REGION Network 11: Output Feedback
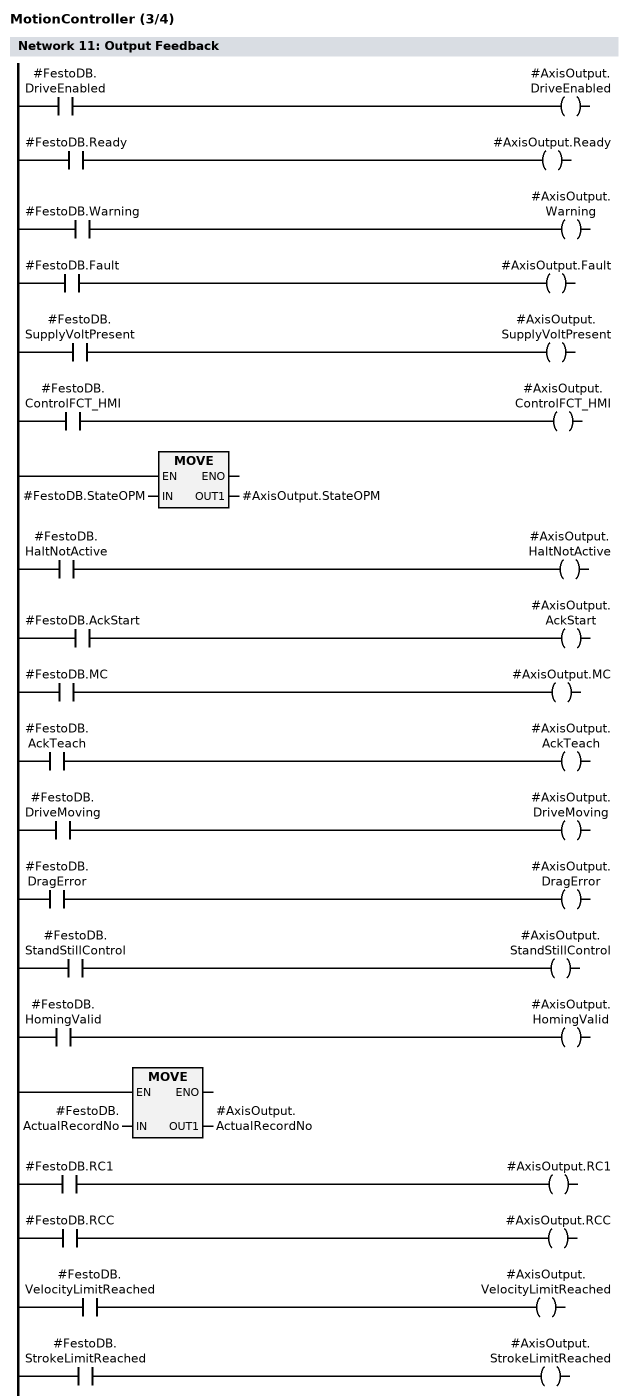
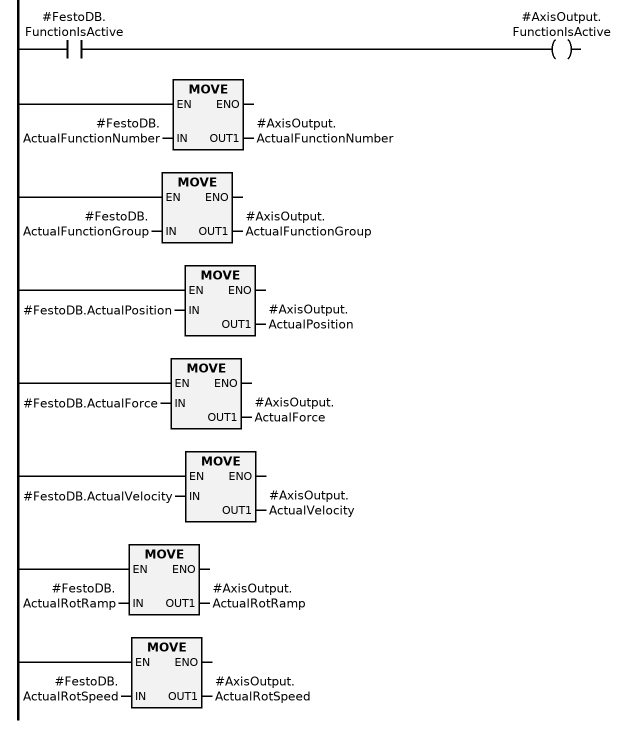
   RUNG wire#powerrail
      Contact( #FestoDB.DriveEnabled )
      Coil( #AxisOutput.DriveEnabled )
   END_RUNG
   RUNG wire#powerrail
      Contact( #FestoDB.Ready )
      Coil( #AxisOutput.Ready )
   END_RUNG
   RUNG wire#powerrail
      Contact( #FestoDB.Warning )
      Coil( #AxisOutput.Warning )
   END_RUNG
   RUNG wire#powerrail
      Contact( #FestoDB.Fault )
      Coil( #AxisOutput.Fault )
   END_RUNG
   RUNG wire#powerrail
      Contact( #FestoDB.SupplyVoltPresent )
      Coil( #AxisOutput.SupplyVoltPresent )
   END_RUNG
   RUNG wire#powerrail
      Contact( #FestoDB.ControlFCT_HMI )
      Coil( #AxisOutput.ControlFCT_HMI )
   END_RUNG
   RUNG wire#powerrail
      Move(in := #FestoDB.StateOPM, out1 => #AxisOutput.StateOPM)
   END_RUNG
   RUNG wire#powerrail
      Contact( #FestoDB.HaltNotActive )
      Coil( #AxisOutput.HaltNotActive )
   END_RUNG
   RUNG wire#powerrail
      Contact( #FestoDB.AckStart )
      Coil( #AxisOutput.AckStart )
   END_RUNG
   RUNG wire#powerrail
      Contact( #FestoDB.MC )
      Coil( #AxisOutput.MC )
   END_RUNG
   RUNG wire#powerrail
      Contact( #FestoDB.AckTeach )
      Coil( #AxisOutput.AckTeach )
   END_RUNG
   RUNG wire#powerrail
      Contact( #FestoDB.DriveMoving )
      Coil( #AxisOutput.DriveMoving )
   END_RUNG
   RUNG wire#powerrail
      Contact( #FestoDB.DragError )
      Coil( #AxisOutput.DragError )
   END_RUNG
   RUNG wire#powerrail
      Contact( #FestoDB.StandStillControl )
      Coil( #AxisOutput.StandStillControl )
   END_RUNG
   RUNG wire#powerrail
      Contact( #FestoDB.HomingValid )
      Coil( #AxisOutput.HomingValid )
   END_RUNG
   RUNG wire#powerrail
      Move(in := #FestoDB.ActualRecordNo, out1 => #AxisOutput.ActualRecordNo)
   END_RUNG
   RUNG wire#powerrail
      Contact( #FestoDB.RC1 )
      Coil( #AxisOutput.RC1 )
   END_RUNG
   RUNG wire#powerrail
      Contact( #FestoDB.RCC )
      Coil( #AxisOutput.RCC )
   END_RUNG
   RUNG wire#powerrail
      Contact( #FestoDB.VelocityLimitReached )
      Coil( #AxisOutput.VelocityLimitReached )
   END_RUNG
   RUNG wire#powerrail
      Contact( #FestoDB.StrokeLimitReached )
      Coil( #AxisOutput.StrokeLimitReached )
   END_RUNG
   RUNG wire#powerrail
      Contact( #FestoDB.FunctionIsActive )
      Coil( #AxisOutput.FunctionIsActive )
   END_RUNG
   RUNG wire#powerrail
      Move(in := #FestoDB.ActualFunctionNumber, out1 => #AxisOutput.ActualFunctionNumber)
   END_RUNG
   RUNG wire#powerrail
      Move(in := #FestoDB.ActualFunctionGroup, out1 => #AxisOutput.ActualFunctionGroup)
   END_RUNG
   RUNG wire#powerrail
      Move(in := #FestoDB.ActualPosition, out1 => #AxisOutput.ActualPosition)
   END_RUNG
   RUNG wire#powerrail
      Move(in := #FestoDB.ActualForce, out1 => #AxisOutput.ActualForce)
   END_RUNG
   RUNG wire#powerrail
      Move(in := #FestoDB.ActualVelocity, out1 => #AxisOutput.ActualVelocity)
   END_RUNG
   RUNG wire#powerrail
      Move(in := #FestoDB.ActualRotRamp, out1 => #AxisOutput.ActualRotRamp)
   END_RUNG
   RUNG wire#powerrail
      Move(in := #FestoDB.ActualRotSpeed, out1 => #AxisOutput.ActualRotSpeed)
   END_RUNG
   // the same network as SCL:
   #AxisOutput.DriveEnabled := #FestoDB.DriveEnabled;
   #AxisOutput.Ready := #FestoDB.Ready;
   #AxisOutput.Warning := #FestoDB.Warning;
   #AxisOutput.Fault := #FestoDB.Fault;
   #AxisOutput.SupplyVoltPresent := #FestoDB.SupplyVoltPresent;
   #AxisOutput.ControlFCT_HMI := #FestoDB.ControlFCT_HMI;
   #AxisOutput.StateOPM := #FestoDB.StateOPM;
   #AxisOutput.HaltNotActive := #FestoDB.HaltNotActive;
   #AxisOutput.AckStart := #FestoDB.AckStart;
   #AxisOutput.MC := #FestoDB.MC;
   #AxisOutput.AckTeach := #FestoDB.AckTeach;
   #AxisOutput.DriveMoving := #FestoDB.DriveMoving;
   #AxisOutput.DragError := #FestoDB.DragError;
   #AxisOutput.StandStillControl := #FestoDB.StandStillControl;
   #AxisOutput.HomingValid := #FestoDB.HomingValid;
   #AxisOutput.ActualRecordNo := #FestoDB.ActualRecordNo;
   #AxisOutput.RC1 := #FestoDB.RC1;
   #AxisOutput.RCC := #FestoDB.RCC;
   #AxisOutput.VelocityLimitReached := #FestoDB.VelocityLimitReached;
   #AxisOutput.StrokeLimitReached := #FestoDB.StrokeLimitReached;
   #AxisOutput.FunctionIsActive := #FestoDB.FunctionIsActive;
   #AxisOutput.ActualFunctionNumber := #FestoDB.ActualFunctionNumber;
   #AxisOutput.ActualFunctionGroup := #FestoDB.ActualFunctionGroup;
   #AxisOutput.ActualPosition := #FestoDB.ActualPosition;
   #AxisOutput.ActualForce := #FestoDB.ActualForce;
   #AxisOutput.ActualVelocity := #FestoDB.ActualVelocity;
   #AxisOutput.ActualRotRamp := #FestoDB.ActualRotRamp;
   #AxisOutput.ActualRotSpeed := #FestoDB.ActualRotSpeed;
END_REGION

REGION Network 12: TargetReached
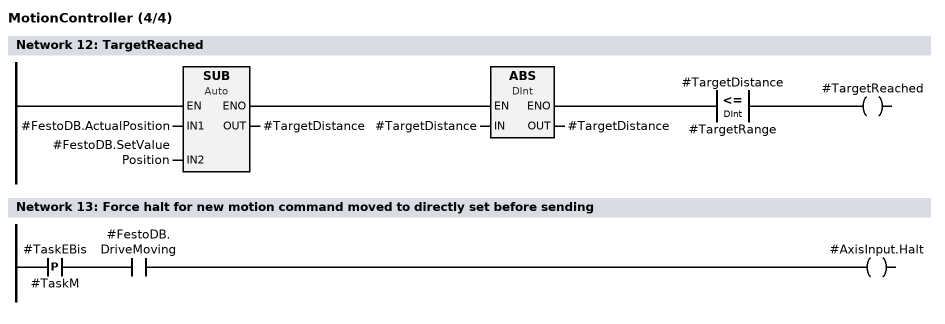
   RUNG wire#powerrail
      Sub(in1 := #FestoDB.ActualPosition, in2 := #FestoDB.SetValuePosition, out => #TargetDistance)
      { S7_Templates := "SrcType := DInt" } Abs(in := #TargetDistance, out => #TargetDistance)
      { S7_Templates := "SrcType := DInt" } LE_Contact(in1 := #TargetDistance, in2 := #TargetRange)
      Coil( #TargetReached )
   END_RUNG
   // the same network as SCL:
   #TargetDistance := #FestoDB.ActualPosition - #FestoDB.SetValuePosition;
   #TargetDistance := ABS(#TargetDistance);
   #TargetReached := #TargetDistance <= #TargetRange;
END_REGION

REGION Network 13: Force halt for new motion command moved to directly set before sending
   RUNG wire#powerrail
      P_Contact(operand := #TaskEBis, bit := #TaskM)
      Contact( #FestoDB.DriveMoving )
      Coil( #AxisInput.Halt )
   END_RUNG
   // the same network as SCL:
   #_w1 := #TaskEBis AND NOT #TaskM;   // rising edge of #TaskEBis
   #TaskM := #TaskEBis;
   #AxisInput.Halt := #_w1 AND #FestoDB.DriveMoving;
END_REGION
END_FUNCTION

FUNCTION_BLOCK "FHPP_DATA_PEEK"
{ S7_Optimized_Access := 'TRUE' }
AUTHOR : FESTO
FAMILY : 'E-DRIVE'
VERSION : 5.3
   VAR_INPUT 
      IAddress_FHPP : Int;
      IAddress_FPC : Int;
      IAdress_FHPPplus : Int;
      DeviceType : String[16];
      cfgFHPPplusIn : DInt;
      SwapBytes : Bool;
   END_VAR

   VAR_OUTPUT 
      Error : Bool;
      Status : "DT_FML_STATUS";
   END_VAR

   VAR_IN_OUT 
      FML_REF : "DT_FML_REF";
   END_VAR

   VAR 
      FHPPplusElementSize : Array[1..9] of DInt;
      FHPPplusSize : DInt;
   END_VAR

   VAR_TEMP 
      tmp_bRetVal : Bool;
      iByteCount : Int;
      i : Int;
      tmpStatus : "DT_FML_STATUS";
      FHPPplus24 : Array[1..24] of Byte;
      tmpFHPPIn : Array[1..16] of Byte;
   END_VAR


BEGIN
	(*############################################################
	    FESTO AG  Co., Esslingen
	    Copyright (c) 2015. All rights reserved.    
	
	    NAME OF FUNCTION BLOCK:         FHPP_DATA_PEEK
	    VERSION NUMBER:                 V5.3
	    COMPOSER:                       bejk
	    
	-----------------------------------------------------
	   Date        Name                Activity                                                                              
	   06.08.2015  Benjamin Kilgus     created (V1.0)
	   15.09.2015  Benjamin Kilgus     errorhandling changed (V1.1)
	   14.10.2015  Benjamin Kilgus     check device type added (V1.2)
	   29.08.2016  Benjamin Klein      version changed (V4.1)
	   20.09.2016  Benjamin Klein      bugfix: FHPPplus and byteorder in FML_REF (V4.2)
	   17.01.2017  Christian Hammer    bugfix: reset variable "tmpStatus" at beginning, label "L_Error" and "L_NO_Error" unified
	   05.07.2017  Benjamin Klein      optimized function block with Slice access instead of AT (V5.1)
	   04.10.2017  Benjamin Klein      devicetype MTR_DCI and SFC_DC added
	   18.10.2017  Benjamin Klein      "tmpStatus" at beginning deleted, labels deleted
	   23.10.2017  Benjamin Klein      SwapBytes Input added for CPX-CM-HPP
	   27.02.2018  Benjamin Klein      Bugfix: Negation of FPC_Mapping in line 75   
	   16.11.2018  Benjamin Klein      Bugfix: Changed tmpFHPPIn from[1..8] to [1..16] (V5.3)
	############################################################*)
	
	// function block (FB) is busy
	#tmpStatus.Err := FALSE;
	#tmpStatus.Cat := 1;
	#tmpStatus.ID := 16#0000_0002; // FB busy
	
	// check device type
	IF #DeviceType = 'CMMO_ST' OR
	    #DeviceType = 'EMCA_EC' OR
	    #DeviceType = 'CMMP_AS' OR
	    #DeviceType = 'CMMS_AS' OR
	    #DeviceType = 'CMMS_ST' OR
	    #DeviceType = 'CMMD_AS' OR
	    #DeviceType = 'SFC_DC' OR
	    #DeviceType = 'MTR_DCI' THEN
	    
	    #FML_REF.DeviceType := #DeviceType;
	ELSE
	    #tmpStatus.Err := TRUE;
	    #tmpStatus.Cat := 1; // functionblock
	    #tmpStatus.ID := DWORD_TO_DINT(16#8000_001E); // device type not valid
	END_IF;
	
	// ### FHPP Standard
	FOR #i := 1 TO 8 DO
	    #FML_REF.InData.FHPP[#i] := PEEK(area := 16#81, dbNumber := 0, byteOffset := #i - 1 + #IAddress_FHPP);
	END_FOR;
	
	// CM-HPP Byte SWAP
	IF #SwapBytes THEN
	    // CM-HPP Byte SWAP
	    #tmpFHPPIn[1] := #FML_REF.InData.FHPP[1];
	    #tmpFHPPIn[2] := #FML_REF.InData.FHPP[2];
	    #tmpFHPPIn[3] := #FML_REF.InData.FHPP[3];
	    #tmpFHPPIn[4] := #FML_REF.InData.FHPP[4];
	    #tmpFHPPIn[5] := #FML_REF.InData.FHPP[8];
	    #tmpFHPPIn[6] := #FML_REF.InData.FHPP[7];
	    #tmpFHPPIn[7] := #FML_REF.InData.FHPP[6];
	    #tmpFHPPIn[8] := #FML_REF.InData.FHPP[5];
	    
	    #FML_REF.InData.FHPP := #tmpFHPPIn;
	    
	END_IF;
	
	
	// ### FPC
	IF #IAddress_FPC <> 0 AND #tmpStatus.Err = FALSE THEN
	    FOR #i := 1 TO 8 DO
	        #FML_REF.InData.FPC[#i] := PEEK(area := 16#81, dbNumber := 0, byteOffset := #i - 1 + #IAddress_FPC);
	    END_FOR;
	    
	    // mapping of FPC data 
	    #tmp_bRetVal := NOT "FPC_MAPPING"(FML_REF := #FML_REF, Mode := FALSE);
	    IF #tmp_bRetVal THEN
	        #tmpStatus.Err := TRUE;
	        #tmpStatus.Cat := 3; // FPC
	        #tmpStatus.ID := 18;
	    END_IF;
	END_IF;
	
	// ### FHPPplus
	IF #IAdress_FHPPplus <> 0 AND #tmpStatus.Err = FALSE THEN
	    
	    // ### check configuration
	    IF #cfgFHPPplusIn <> 0 THEN
	        
	        #tmpStatus.ID := "FHPPPLUS_MAPPING"(cfgFHPPplus := #cfgFHPPplusIn, FHPPplusElementSize => #FHPPplusElementSize, FHPPplusSize => #FHPPplusSize);
	        
	        // FHPP+ Berechnung fehlerhaft beendet
	        IF #tmpStatus.ID <> 0 THEN
	            #tmpStatus.Err := TRUE;
	            #tmpStatus.Cat := 1; // functionblock
	        END_IF;
	    END_IF;
	    
	    #FHPPplusSize := #FHPPplusSize / 8;
	    FOR #i := 1 TO #FHPPplusSize DO
	        #FHPPplus24[#i] := PEEK(area := 16#81, dbNumber := 0, byteOffset := #i - 1 + #IAdress_FHPPplus);
	    END_FOR;
	    
	    
	    
	    // copy data into FML_REF
	    #iByteCount := 1;
	    FOR #i := 1 TO 9 DO
	        CASE #FHPPplusElementSize[#i] OF
	            0:(* Element is empty *)
	                #FML_REF.InData.FHPPplus[#i] := 0;
	                #iByteCount := #iByteCount + 1;
	            8:(* Element is a BYTE *)
	                #FML_REF.InData.FHPPplus[#i] := #FHPPplus24[#iByteCount];
	                #iByteCount := #iByteCount + 1;
	            16:(* Element is a WORD *)
	                #FML_REF.InData.FHPPplus[#i].%B1 := #FHPPplus24[#iByteCount];
	                #FML_REF.InData.FHPPplus[#i].%B0 := #FHPPplus24[#iByteCount + 1];
	                #iByteCount := #iByteCount + 2;
	                
	            32:(* Element is a DWORD *)
	                #FML_REF.InData.FHPPplus[#i].%B3 := #FHPPplus24[#iByteCount];
	                #FML_REF.InData.FHPPplus[#i].%B2 := #FHPPplus24[#iByteCount + 1];
	                #FML_REF.InData.FHPPplus[#i].%B1 := #FHPPplus24[#iByteCount + 2];
	                #FML_REF.InData.FHPPplus[#i].%B0 := #FHPPplus24[#iByteCount + 3];
	                #iByteCount := #iByteCount + 4;
	        END_CASE;
	    END_FOR;
	END_IF;
	
	// ### EXIT ROUTINE ############################################################
	IF NOT #tmpStatus.Err THEN
	    ENO := TRUE;      // Set ENO-Bit to true
	    #Status := #tmpStatus;
	    #Error := #tmpStatus.Err;
	ELSE
	    ENO := FALSE;     // Set ENO-Bit to false
	    #Status := #tmpStatus;
	    #Error := #tmpStatus.Err;
	END_IF;
END_FUNCTION_BLOCK

FUNCTION_BLOCK "FHPP_DATA_POKE"
{ S7_Optimized_Access := 'TRUE' }
AUTHOR : FESTO
FAMILY : 'E-DRIVE'
VERSION : 5.3
   VAR_INPUT 
      OAddress_FHPP : Int;
      OAddress_FPC : Int;
      OAddress_FHPPplus : Int;
      cfgFHPPplusOut : DInt;
      SwapBytes : Bool;
   END_VAR

   VAR_OUTPUT 
      Error : Bool;
      Status : "DT_FML_STATUS";
   END_VAR

   VAR_IN_OUT 
      FML_REF : "DT_FML_REF";
   END_VAR

   VAR 
      FHPPplusElementSize : Array[1..9] of DInt;
      FHPPplusSize : DInt;
      tmpStatus : "DT_FML_STATUS";
   END_VAR

   VAR_TEMP 
      tmp_bRetVal : Bool;
      iByteCount : Int;
      i : Int;
      tmpSize : DInt;
      FHPPplus24 : Array[1..24] of Byte;
      tmpFHPPOut : Array[1..16] of Byte;
   END_VAR


BEGIN
	(*############################################################
	    FESTO AG  Co., Esslingen
	    Copyright (c) 2015. All rights reserved.    
	
	    NAME OF FUNCTION BLOCK:         FHPP_DATA_POKE
	    VERSION NUMBER:                 V5.3
	    COMPOSER:                       bejk
	    
	    -----------------------------------------------------
	   Date        Name                Activity                                                                              
	   06.08.2015  Benjamin Kilgus     created (V1.0)
	   15.09.2015  Benjamin Kilgus     errorhandling changed (V1.1)
	   11.08.2016  Benjamin Klein      bugfix in copy data, first copy then write to output (V1.2)
	   29.08.2016  Benjamin Klein      version changed (V4.1)
	   20.09.2016  Benjamin Klein      Bugfix: byteorder in FML_REF changed and FHPPPlus (V4.2)
	   17.01.2017  Christian Hammer    bugfix: reset variable "tmpStatus" at beginning, label "L_Error" and "L_NO_Error" unified
	   05.07.2017  Benjamin Klein      optimized function block with Slice access instead of AT (V5.1)
	   18.10.2017  Benjamin Klein      "tmpStatus" at beginning deleted, labels deleted
	   23.10.2017  Benjamin Klein      SwapBytes Input added for CPX-CM-HPP
	   27.02.2018  Benjamin Klein      Bugfix: Negation of FPC_Mapping in line 78 
	   16.11.2018  Benjamin Klein      Bugfix: Changed tmpFHPPIn from[1..8] to [1..16] (V5.3)
	############################################################*)
	
	// function block (FB) is busy
	#tmpStatus.Err := FALSE;
	#tmpStatus.Cat := 1;
	#tmpStatus.ID := 16#0000_0002; // FB busy
	
	// CM-HPP Byte SWAP
	IF #SwapBytes THEN
	    #tmpFHPPOut[1] := #FML_REF.OutData.FHPP[1];
	    #tmpFHPPOut[2] := #FML_REF.OutData.FHPP[2];
	    #tmpFHPPOut[3] := #FML_REF.OutData.FHPP[3];
	    #tmpFHPPOut[4] := #FML_REF.OutData.FHPP[4];
	    #tmpFHPPOut[5] := #FML_REF.OutData.FHPP[8];
	    #tmpFHPPOut[6] := #FML_REF.OutData.FHPP[7];
	    #tmpFHPPOut[7] := #FML_REF.OutData.FHPP[6];
	    #tmpFHPPOut[8] := #FML_REF.OutData.FHPP[5];
	    
	    #FML_REF.OutData.FHPP := #tmpFHPPOut;
	END_IF;
	
	
	// copy data into FML_REF
	#iByteCount := 1;
	FOR #i := 1 TO 9 DO
	    CASE #FHPPplusElementSize[#i] OF
	        0:(* Element is empty *)
	            #FML_REF.OutData.FHPPplus[#i] := 0;
	            #iByteCount := #iByteCount + 1;
	        8:(* Element is a BYTE *)
	            #FHPPplus24[#iByteCount] := #FML_REF.OutData.FHPPplus[#i];
	            #iByteCount := #iByteCount + 1;
	        16:(* Element is a WORD *)
	            #FHPPplus24[#iByteCount] := #FML_REF.OutData.FHPPplus[#i].%B1;
	            #FHPPplus24[#iByteCount + 1] := #FML_REF.OutData.FHPPplus[#i].%B0;
	            #iByteCount := #iByteCount + 2;
	        32:(* Element is a DWORD *)
	            #FHPPplus24[#iByteCount] := #FML_REF.OutData.FHPPplus[#i].%B3;
	            #FHPPplus24[#iByteCount + 1] := #FML_REF.OutData.FHPPplus[#i].%B2;
	            #FHPPplus24[#iByteCount + 2] := #FML_REF.OutData.FHPPplus[#i].%B1;
	            #FHPPplus24[#iByteCount + 3] := #FML_REF.OutData.FHPPplus[#i].%B0;
	            #iByteCount := #iByteCount + 4;
	    END_CASE;
	END_FOR;
	
	
	// ### FHPP Data
	FOR #i := 1 TO 8 DO
	    POKE(area := 16#82,
	         dbNumber := 0,
	         byteOffset := #i - 1 + #OAddress_FHPP,
	         value := #FML_REF.OutData.FHPP[#i]);
	END_FOR;
	
	// ### FPC Data
	IF #OAddress_FPC <> 0 AND #tmpStatus.Err = FALSE THEN
	    // mapping of FPC data 
	    #tmp_bRetVal := NOT "FPC_MAPPING"(FML_REF := #FML_REF, Mode := TRUE);
	    IF #tmp_bRetVal THEN
	        #tmpStatus.Err := TRUE;
	        #tmpStatus.Cat := 3; // FPC
	        #tmpStatus.ID := 18;
	    END_IF;
	    
	    FOR #i := 1 TO 8 DO
	        POKE(area := 16#82,
	             dbNumber := 0,
	             byteOffset := #i - 1 + #OAddress_FPC,
	             value := #FML_REF.OutData.FPC[#i]);
	    END_FOR;
	END_IF;
	
	
	// ### FHPP PLUS Data
	
	
	IF #OAddress_FHPPplus <> 0 AND #tmpStatus.Err = FALSE THEN
	    
	    // check configuration  
	    IF #cfgFHPPplusOut <> 0 THEN
	        #tmpStatus.ID := "FHPPPLUS_MAPPING"(cfgFHPPplus := #cfgFHPPplusOut, FHPPplusElementSize => #FHPPplusElementSize, FHPPplusSize => #FHPPplusSize);
	        // FHPP+ Berechnung fehlerhaft beendet
	        IF #tmpStatus.ID <> 0 THEN
	            #tmpStatus.Err := TRUE;
	            #tmpStatus.Cat := 1; // functionblock
	        END_IF;
	    END_IF;
	    
	    #FHPPplusSize := #FHPPplusSize / 8;
	    
	    FOR #i := 1 TO #FHPPplusSize DO
	        POKE(area := 16#82,
	             dbNumber := 0,
	             byteOffset := #i - 1 + #OAddress_FHPPplus,
	             value := #FHPPplus24[#i]);
	    END_FOR;
	END_IF;
	
	// ### EXIT ROUTINE ############################################################
	IF NOT #tmpStatus.Err THEN
	    ENO := TRUE;      // Set ENO-Bit to true
	    #Status := #tmpStatus;
	    #Error := #tmpStatus.Err;
	ELSE
	    ENO := FALSE;     // Set ENO-Bit to false
	    #Status := #tmpStatus;
	    #Error := #tmpStatus.Err;
	END_IF;
END_FUNCTION_BLOCK

FUNCTION_BLOCK "FPC_DIAG"
{ S7_Optimized_Access := 'TRUE' }
AUTHOR : FESTO
FAMILY : 'E-DRIVE'
VERSION : 5.3
   VAR_INPUT 
      Execute : Bool;
   END_VAR

   VAR_OUTPUT 
      Done : Bool;
      Error : Bool;
      MessageNumber : DInt;
      Status : "DT_FML_STATUS";
   END_VAR

   VAR_IN_OUT 
      FML_REF : "DT_FML_REF";
   END_VAR

   VAR 
      bInit : Bool := FALSE;
      TimeStart : Bool;
      lMemberID : Int := 0;
      tmpDevice : String[16];
      TONinst {InstructionName := 'TON_TIME'; LibVersion := '1.0'} : TON_TIME;
      tmpStatus { ExternalAccessible := 'False'; ExternalVisible := 'False'; ExternalWritable := 'False'} : "DT_FML_STATUS";
   END_VAR

   VAR CONSTANT 
      TimeoutTime : Time := T#3S;
   END_VAR


BEGIN
	(*############################################################
	   FESTO AG  Co., Essling
	   
	   Copyright (c) 2015. All rights reserved.    
	
	   NAME OF FUNCTION BLOCK:         FPC_DIAG
	   VERSION NUMBER:                 V5.3
	   COMPOSER:                       bejk
	   
	   -----------------------------------------------------
	   Date        Name                Activity                                                                              
	   06.08.2015  Benjamin Kilgus     created (V1.0)
	   20.08.2015  Benjamin Kilgus     Timeout logic added (V1.1)
	   14.09.2015  Benjamin Kilgus     error handling changed (V1.2)
	   16.11.2015  Benjamin Kilgus     Option optimierter Baustein Zugriff entfernt (V1.3)
	   29.08.2016  Benjamin Klein      version changed (V4.1)
	   17.01.2017  Christian Hammer    bugfix: reset variable "tmpStatus" at beginning
	                                   changed condition in ASSIGNMENT OF STATUS from "Status.Err" to "tmpStatus.Err"
	   21.02.2017  Benjamin Klein      added GoTo Error if Error occurs, Labels added
	   05.07.2017  Benjamin Klein      optimized access added (V5.1)
	   04.10.2017  Benjamin Klein      devicetype MTR_DCI and SFC_DC added
	   18.10.2017  Benjamin Klein      "tmpStatus" at beginning deleted, labels deleted
	   16.04.2018  Benjamin Klein      CMXH-ST added (V5.3)
	############################################################*)
	
	(* ====== initial block routine ===================================== *)
	(* ----- get MemberID for this function block ------------------------*)
	IF NOT #bInit THEN
	    #FML_REF.MemberIDmax := #FML_REF.MemberIDmax + 1;
	    #lMemberID := #FML_REF.MemberIDmax;
	    #Status.Err := FALSE;
	    #Status.Cat := 1; // Functionblock
	    #Status.ID := 16#0000_0001;
	    #bInit := TRUE;
	    RETURN;
	END_IF;
	
	(* ====== supervision of timeout ==================================== *)
	(* ----- timer to monitor a timeout of the function block ------------*)
	#TONinst(IN := #TimeStart,
	         PT := #TimeoutTime);
	IF #TONinst.Q THEN
	    #Done := TRUE;
	    #tmpStatus.Err := TRUE;
	    #tmpStatus.Cat := 1;
	    #tmpStatus.ID := DWORD_TO_DINT(16#8000_0014); // FB timeout
	END_IF;
	
	(* ===== logic part ================================================= *)
	(* ----- ASSIGNMENT OF STATUS --------------------------------------- *)
	IF #FML_REF.MemberID = #lMemberID AND #tmpStatus.ID <> DWORD_TO_DINT(16#8000_001E) THEN
	    IF #FML_REF.Done AND NOT #FML_REF.Err AND NOT #tmpStatus.Err THEN
	        #Done := TRUE;
	        #TimeStart := FALSE;
	        IF #FML_REF.ParamValueRD = 65535 THEN // special: -1 to 0
	            #MessageNumber := 0;
	        ELSE
	            #MessageNumber := #FML_REF.ParamValueRD;
	        END_IF;
	        
	        #tmpStatus.Err := FALSE;
	        #tmpStatus.Cat := 0;
	        #tmpStatus.ID := 16#0000_0000;
	        
	    ELSIF #FML_REF.Err THEN
	        #tmpStatus.Err := TRUE;
	        #tmpStatus.Cat := 3;
	        #tmpStatus.ID := #FML_REF.ParamValueRD;
	    END_IF;
	END_IF;
	
	(* ----- ASSIGNMENT OF CONTROL at rising edge of Execute ------------ *)
	IF (#FML_REF.MemberID = 0) AND #Execute AND NOT #tmpStatus.Err THEN
	    #FML_REF.MemberID := #lMemberID;
	    #FML_REF.ReqID := 6; // read array dword
	    #TimeStart := TRUE;
	    #tmpStatus.Err := FALSE;
	    #tmpStatus.Cat := 1; // Functionblock
	    #tmpStatus.ID := 16#0000_0002; // FB busy    
	    
	    #tmpDevice := #FML_REF.DeviceType;
	    
	    IF #tmpDevice = 'EMCA_EC' OR #tmpDevice = 'CMMO_ST' OR #tmpDevice = 'CMXH_ST' THEN
	        #FML_REF.FPCC_Modus := 1; // EFPC enhanced
	        #FML_REF.PNU := 205;
	        #FML_REF.Subindex := 1;
	    ELSIF #tmpDevice = 'SFC_DC' OR #tmpDevice = 'MTR_DCI' THEN
	        #Done := TRUE;
	        #tmpStatus.Err := TRUE;
	        #tmpStatus.Cat := 1;
	        #tmpStatus.ID := DWORD_TO_DINT(16#8000_001E); // wrong Device Type
	        #TimeStart := FALSE;
	    ELSE
	        #FML_REF.FPCC_Modus := 0; // FPC Standard
	        #FML_REF.PNU := 201;
	        #FML_REF.Subindex := 1;
	    END_IF;
	    
	ELSIF (#FML_REF.MemberID = #lMemberID) AND NOT #Execute THEN
	    #FML_REF.ReqID := 0; // none request
	    #FML_REF.FPCC_Modus := 0;
	    #FML_REF.PNU := 0;
	    #FML_REF.Subindex := 0;
	    #FML_REF.ParamValueWR := 0;
	    #TimeStart := TRUE;
	    #MessageNumber := 0;
	    
	    // release access if done is false
	    IF NOT #FML_REF.Done THEN
	        #FML_REF.MemberID := 0;
	        #Done := FALSE;
	        #TimeStart := FALSE;
	        #tmpStatus.Err := FALSE;
	        #tmpStatus.Cat := 0;
	        #tmpStatus.ID := 16#0000_0000;
	    END_IF;
	    
	ELSIF (#FML_REF.MemberID <> #lMemberID) AND NOT #tmpStatus.Err THEN
	    IF #Execute THEN
	        #tmpStatus.Err := FALSE;
	        #tmpStatus.Cat := 1;
	        #tmpStatus.ID := 16#0000_000A; // other FB active
	    ELSE
	        #tmpStatus.Err := FALSE;
	        #tmpStatus.Cat := 0;
	        #tmpStatus.ID := 16#0000_0000;
	    END_IF;
	END_IF;
	
	// ### EXIT ROUTINE ############################################################
	IF NOT #tmpStatus.Err THEN
	    ENO := TRUE;      // Set ENO-Bit to true
	    #Status := #tmpStatus;
	    #Error := #tmpStatus.Err;
	ELSE
	    ENO := FALSE;     // Set ENO-Bit to false
	    #Status := #tmpStatus;
	    #Error := #tmpStatus.Err;
	END_IF;
	
END_FUNCTION_BLOCK

FUNCTION_BLOCK "FPC_PNU"
{ S7_Optimized_Access := 'TRUE' }
AUTHOR : FESTO
FAMILY : 'E-DRIVE'
VERSION : 5.1
   VAR_INPUT 
      Execute : Bool;
      Write : Bool;
      DatatypeWR : Int;
      PNU : Word;
      Subindex : Byte;
      Value : DInt;
   END_VAR

   VAR_OUTPUT 
      Done : Bool;
      Error : Bool;
      ActPNU : Word;
      ActSubindex : Byte;
      ActValue : DInt;
   END_VAR
   VAR_OUTPUT DB_SPECIFIC
      DatatypeRD : Int;
   END_VAR
   VAR_OUTPUT 
      Status : "DT_FML_STATUS";
   END_VAR

   VAR_IN_OUT 
      FML_REF : "DT_FML_REF";
   END_VAR

   VAR 
      bInit : Bool := FALSE;
      TimeStart : Bool;
      lMemberID : Int := 0;
      tmpDevice : String[16];
      TONInst {InstructionName := 'TON_TIME'; LibVersion := '1.0'} : TON_TIME;
      tmpStatus : "DT_FML_STATUS";
   END_VAR

   VAR CONSTANT 
      TimeoutTime : Time := T#3S;
   END_VAR


BEGIN
	(*############################################################
	   FESTO AG  Co., Esslingen
	   Copyright (c) 2015. All rights reserved.    
	
	   NAME OF FUNCTION BLOCK:         FPC_PNU
	   VERSION NUMBER:                 V5.1
	   COMPOSER:                       bejk
	  
	  
	   -----------------------------------------------------
	   Date        Name                Activity                                                                              
	   06.08.2015  Benjamin Kilgus     created (V1.0)
	   20.08.2015  Benjamin Kilgus     Timeout logic added (V1.1)
	   07.09.2015  Benjamin Kilgus     error handling changed (V1.2)
	   28.10.2015  Benjamin Kilgus     Timeout beim wegnehmen von Execute nicht abprüfen wegen bug im CMMP (V1.3)
	   16.11.2015  Benjamin Kilgus     Zeile 36 --> #Status.Err := TRUE;
	                                   Zeile 97 --> #TimeStart := FALSE;
	                                   Option optimierter Baustein Zugriff entfernt (V1.4)      
	   29.08.2016  Benjamin Klein      version changed (V4.1)
	   19.10.2016  Benjamin Klein      Set ActValue in case of error to 0, tmpStatus Error fixed (V4.2)
	   18.04.2017  Benjamin Klein      optimized access (V5.1)
	   04.10.2017  Benjamin Klein      devicetype MTR_DCI and SFC_DC added
	   20.11.2017  Benjamin Klein      copy the DataypeRD and DataypeWR(MTR and SFC only)
	############################################################*)
	
	(* ====== initial block routine ===================================== *)
	(* ----- get MemberID for this function block ------------------------*)
	IF NOT #bInit THEN
	    #FML_REF.MemberIDmax := #FML_REF.MemberIDmax + 1;
	    #lMemberID := #FML_REF.MemberIDmax;
	    #bInit := TRUE;
	    #Status.Err := False;
	    #Status.Cat := 1;
	    #Status.ID := 1; // init active     
	    RETURN;
	END_IF;
	
	(* ====== supervision of timeout ==================================== *)
	(* ----- timer to monitor a timeout of the function block ------------*)
	// Timout Timer
	#TONInst(IN := #TimeStart,
	         PT := #TimeoutTime);
	
	IF #TONInst.Q THEN
	    #Done := TRUE;
	    #tmpStatus.Err := TRUE;
	    #tmpStatus.Cat := 1;
	    #tmpStatus.ID := DWORD_TO_DINT(16#8000_0014); // FB timeout         
	END_IF;
	
	(* ===== logic part ================================================= *)
	(* ----- ASSIGNMENT OF STATUS --------------------------------------- *)
	IF #FML_REF.MemberID = #lMemberID THEN
	    IF #FML_REF.Done AND NOT #tmpStatus.Err THEN
	        #TimeStart := False;
	        #Done := True;
	        #ActSubindex := #FML_REF.ActSubindex;
	        #ActPNU := #FML_REF.ActPNU;
	        #ActValue := #FML_REF.ParamValueRD;
	        #DatatypeRD := #FML_REF.DatatypeRD;
	        #tmpStatus.Err := False;
	        #tmpStatus.Cat := 0;
	        #tmpStatus.ID := 0; // none    
	        IF #FML_REF.Err THEN
	            #tmpStatus.Err := TRUE;
	            #tmpStatus.Cat := 3;
	            #tmpStatus.ID := #FML_REF.ParamValueRD; // FPC error
	            #ActValue := 0;
	        END_IF;
	    END_IF;
	END_IF;
	
	(* ----- ASSIGNMENT OF CONTROL at rising edge of execute ----------- *)
	IF (#FML_REF.MemberID = 0) AND #Execute THEN
	    #FML_REF.MemberID := #lMemberID;
	    #TimeStart := TRUE;
	    #tmpStatus.Err := FALSE;
	    #tmpStatus.Cat := 1;
	    #tmpStatus.ID := 16#0000_00002; // busy 
	    
	    #FML_REF.PNU := #PNU;
	    #FML_REF.Subindex := #Subindex;
	    #FML_REF.ParamValueWR := #Value;
	    
	    IF #Write THEN
	        #FML_REF.DatatypeWR := INT_TO_BYTE(#DatatypeWR);
	        #FML_REF.ReqID := 8; // write array dword        
	    ELSE
	        #FML_REF.ReqID := 6; //read array 
	    END_IF;
	    
	    #tmpDevice := #FML_REF.DeviceType;
	    IF #tmpDevice = 'EMCA_EC' OR #tmpDevice = 'CMMO_ST' THEN
	        #FML_REF.FPCC_Modus := 1; // EFPC enhanced
	    ELSE
	        #FML_REF.FPCC_Modus := 0; // FPC Standard
	    END_IF;
	    
	ELSIF (#FML_REF.MemberID = #lMemberID) AND NOT #Execute THEN
	    #FML_REF.ReqID := 0;
	    #FML_REF.FPCC_Modus := 0;
	    #FML_REF.PNU := 0;
	    #FML_REF.Subindex := 0;
	    #FML_REF.ParamValueWR := 0;
	    #ActSubindex := 0;
	    #ActPNU := 0;
	    #ActValue := 0;
	    //TimeStart         := TRUE;            (* BUG IN FIRMWARE CMMP_AS (V4.0.10.1501.13.61) --> Zeile in Lib derzeit nicht umsetzbar --> Problem am 14.09.2015 gemeldet (CHMM) *)
	    IF NOT #FML_REF.Done THEN
	        #FML_REF.FPCC_Modus := 0;
	        #FML_REF.MemberID := 0;
	        #Done := FALSE;
	        #TimeStart := FALSE;
	        #tmpStatus.Err := FALSE;
	        #tmpStatus.Cat := 0;
	        #tmpStatus.ID := 16#0000_00000; // none 
	    END_IF;
	    
	ELSIF (#FML_REF.MemberID <> #lMemberID) THEN
	    IF #Execute THEN
	        #tmpStatus.Err := FALSE;
	        #tmpStatus.Cat := 1;
	        #tmpStatus.ID := 16#0000_0000A; // other FB active
	    ELSE
	        #tmpStatus.Err := FALSE;
	        #tmpStatus.Cat := 0;
	        #tmpStatus.ID := 0; // none
	    END_IF;
	END_IF;
	
	#Error := #tmpStatus.Err;
	#Status := #tmpStatus;
END_FUNCTION_BLOCK

DATA_BLOCK "Capping_Station_DB"   // DB15
VERSION : 0.1
"Capping_Station"
BEGIN
END_DATA_BLOCK

DATA_BLOCK "Heater_Control_DB"   // DB37
VERSION : 0.1
"IR_Heater_Control"
BEGIN
END_DATA_BLOCK

DATA_BLOCK "LED_Behavior_DB"   // DB51
VERSION : 0.1
"LED_Behavior"
BEGIN
END_DATA_BLOCK

DATA_BLOCK "LoadCell_FluidTankWeight_DB"   // DB23
VERSION : 0.1
"LoadCell"
BEGIN
END_DATA_BLOCK

DATA_BLOCK "LoadCell_WasteTankWeight_DB"   // DB31
VERSION : 0.1
"LoadCell"
BEGIN
END_DATA_BLOCK

DATA_BLOCK "RollerV3_DB"   // DB10
VERSION : 0.1
"RollerV3"
BEGIN
END_DATA_BLOCK

DATA_BLOCK "AXIS_X_Motion_V2_Festo_PtP_Drives_PN_DB"   // DB28
AUTHOR : Festo
FAMILY : E-.Drives
VERSION : 1.5
"Festo_PtP_Drives_PN"
BEGIN
END_DATA_BLOCK

DATA_BLOCK "AXIS_X_V2_CMMT"   // DB8
VERSION : 0.1
"AXIS_CMMT_V2_Motion_Control"
BEGIN
END_DATA_BLOCK

DATA_BLOCK "AXIS_Y_Motion_V2_Festo_PtP_Drives_PN_DB"   // DB1
AUTHOR : Festo
FAMILY : E-.Drives
VERSION : 1.5
"Festo_PtP_Drives_PN"
BEGIN
END_DATA_BLOCK

DATA_BLOCK "AXIS_Y_V2_CMMT"   // DB29
VERSION : 0.1
"AXIS_CMMT_V2_Motion_Control"
BEGIN
END_DATA_BLOCK

DATA_BLOCK "AXIS_Z1_Motion_V2_Festo_PtP_Drives_PN_DB"   // DB3
AUTHOR : Festo
FAMILY : E-.Drives
VERSION : 1.5
"Festo_PtP_Drives_PN"
BEGIN
END_DATA_BLOCK

DATA_BLOCK "AXIS_Z1_V2_CMMT"   // DB40
VERSION : 0.1
"AXIS_CMMT_V2_Motion_Control"
BEGIN
END_DATA_BLOCK

DATA_BLOCK "AXIS_Z2_Motion_V2_Festo_PtP_Drives_PN_DB"   // DB39
AUTHOR : Festo
FAMILY : E-.Drives
VERSION : 1.5
"Festo_PtP_Drives_PN"
BEGIN
END_DATA_BLOCK

DATA_BLOCK "AXIS_Z2_V2_CMMT"   // DB41
VERSION : 0.1
"AXIS_CMMT_V2_Motion_Control"
BEGIN
END_DATA_BLOCK

DATA_BLOCK "CMMS_Z1_Movement_DB"   // DB76
VERSION : 0.1
"CMMS_Z1_Movement"
BEGIN
END_DATA_BLOCK

DATA_BLOCK "CMMS_Z2_Movement_DB"   // DB77
VERSION : 0.1
"CMMS_Z2_Movement"
BEGIN
END_DATA_BLOCK

DATA_BLOCK "Initial_Test_Squence_DB"   // DB78
VERSION : 0.1
"Initial_Test_Squence"
BEGIN
END_DATA_BLOCK

DATA_BLOCK "Stacklight_DB"   // DB83
VERSION : 0.1
"Stacklight"
BEGIN
END_DATA_BLOCK

DATA_BLOCK "UVLamp_DB"   // DB82
VERSION : 0.1
"UVLamp"
BEGIN
END_DATA_BLOCK

DATA_BLOCK "Z axis missing layer detection_DB"   // DB101
VERSION : 0.1
"Z axis missing layer detection"
BEGIN
END_DATA_BLOCK

DATA_BLOCK "AXIS_Z1_V2_CMMS"   // DB66
VERSION : 0.1
"AXIS_CMMT_V2_Motion_Control"
BEGIN
END_DATA_BLOCK

DATA_BLOCK "AXIS_Z2_V2_CMMS"   // DB72
VERSION : 0.1
"AXIS_CMMT_V2_Motion_Control"
BEGIN
END_DATA_BLOCK

DATA_BLOCK "CMMS_Z1_FHPP_CTRL_DB"   // DB70
AUTHOR : FESTO
FAMILY : E-DRIVE
VERSION : 5.1
"FHPP_CTRL"
BEGIN
END_DATA_BLOCK

DATA_BLOCK "CMMS_Z1_FHPP_DPRD_DAT_DB"   // DB67
AUTHOR : FESTO
FAMILY : E-DRIVE
VERSION : 5.1
"FHPP_DPRD_DAT"
BEGIN
END_DATA_BLOCK

DATA_BLOCK "CMMS_Z1_FHPP_DPWR_DAT_DB"   // DB71
AUTHOR : FESTO
FAMILY : E-DRIVE
VERSION : 5.1
"FHPP_DPWR_DAT"
BEGIN
END_DATA_BLOCK

DATA_BLOCK "CMMS_Z2_FHPP_CTRL_DB"   // DB74
AUTHOR : FESTO
FAMILY : E-DRIVE
VERSION : 5.1
"FHPP_CTRL"
BEGIN
END_DATA_BLOCK

DATA_BLOCK "CMMS_Z2_FHPP_DPRD_DAT_DB"   // DB73
AUTHOR : FESTO
FAMILY : E-DRIVE
VERSION : 5.1
"FHPP_DPRD_DAT"
BEGIN
END_DATA_BLOCK

DATA_BLOCK "CMMS_Z2_FHPP_DPWR_DAT_DB"   // DB75
AUTHOR : FESTO
FAMILY : E-DRIVE
VERSION : 5.1
"FHPP_DPWR_DAT"
BEGIN
END_DATA_BLOCK

DATA_BLOCK "NoGoZoneV1_01_DB"   // DB86
VERSION : 0.1
"NoGoZoneV1"
BEGIN
END_DATA_BLOCK

DATA_BLOCK "Control_Buttons_Activation_DB"   // DB89
VERSION : 0.1
"Control_Buttons_Activation"
BEGIN
END_DATA_BLOCK

DATA_BLOCK "Control_Buttons_Manipulate_DB"   // DB90
VERSION : 0.1
"Control_Buttons_Manipulate"
BEGIN
END_DATA_BLOCK

DATA_BLOCK "DataLogging_DB"   // DB94
VERSION : 0.1
"DataLogging"
BEGIN
END_DATA_BLOCK

DATA_BLOCK "ZAxis_RelativeMotion_Test_DB"   // DB96
VERSION : 0.1
"ZAxis_RelativeMotion_Test"
BEGIN
END_DATA_BLOCK

DATA_BLOCK "BlinkTimer"   // DB20
{ S7_Optimized_Access := 'TRUE' }
"IEC_TIMER"
   // VAR
   //    PT : Time;
   //    ET : Time;
   //    IN : Bool;
   //    Q : Bool;
   // END_VAR
BEGIN
END_DATA_BLOCK

DATA_BLOCK "Buttons_Homing_Delay"   // DB93
{ S7_Optimized_Access := 'TRUE' }
"IEC_TIMER"
   // VAR
   //    PT : Time;
   //    ET : Time;
   //    IN : Bool;
   //    Q : Bool;
   // END_VAR
BEGIN
END_DATA_BLOCK

DATA_BLOCK "CTRL_PWM_DB"   // DB32
"CTRL_PWM_SFB"
   // VAR_INPUT
   //    PWM : HW_PWM;
   //    ENABLE : Bool;
   // END_VAR
   // VAR_OUTPUT
   //    BUSY : Bool;
   //    STATUS : Word;
   // END_VAR
BEGIN
END_DATA_BLOCK

DATA_BLOCK "CappingStationSafety"   // DB59
{ S7_Optimized_Access := 'TRUE' }
"IEC_TIMER"
   // VAR
   //    PT : Time;
   //    ET : Time;
   //    IN : Bool;
   //    Q : Bool;
   // END_VAR
BEGIN
END_DATA_BLOCK

DATA_BLOCK "CappingStationTest01"   // DB48
{ S7_Optimized_Access := 'TRUE' }
"IEC_TIMER"
   // VAR
   //    PT : Time;
   //    ET : Time;
   //    IN : Bool;
   //    Q : Bool;
   // END_VAR
BEGIN
END_DATA_BLOCK

DATA_BLOCK "CappingStationTest02"   // DB52
{ S7_Optimized_Access := 'TRUE' }
"IEC_TIMER"
   // VAR
   //    PT : Time;
   //    ET : Time;
   //    IN : Bool;
   //    Q : Bool;
   // END_VAR
BEGIN
END_DATA_BLOCK

DATA_BLOCK "CappingStation_CounterNEW"   // DB62
{ S7_Optimized_Access := 'TRUE' }
"IEC_COUNTER"
   // VAR RETAIN
   //    CU : Bool;
   //    CD : Bool;
   //    R : Bool;
   //    LD : Bool;
   //    QU : Bool;
   //    QD : Bool;
   //    PV : Int;
   //    CV : Int;
   // END_VAR
BEGIN
END_DATA_BLOCK

DATA_BLOCK "CappingStation_CounterON"   // DB61
{ S7_Optimized_Access := 'TRUE' }
"IEC_DCOUNTER"
   // VAR RETAIN
   //    CU : Bool;
   //    CD : Bool;
   //    R : Bool;
   //    LD : Bool;
   //    QU : Bool;
   //    QD : Bool;
   //    PV : DInt;
   //    CV : DInt;
   // END_VAR
BEGIN
END_DATA_BLOCK

DATA_BLOCK "Control_Buttons_OFFdelay_DB"   // DB91
{ S7_Optimized_Access := 'TRUE' }
"IEC_TIMER"
   // VAR
   //    PT : Time;
   //    ET : Time;
   //    IN : Bool;
   //    Q : Bool;
   // END_VAR
BEGIN
END_DATA_BLOCK

DATA_BLOCK "Control_Buttons_Read_Delay"   // DB92
{ S7_Optimized_Access := 'TRUE' }
"IEC_TIMER"
   // VAR
   //    PT : Time;
   //    ET : Time;
   //    IN : Bool;
   //    Q : Bool;
   // END_VAR
BEGIN
END_DATA_BLOCK

DATA_BLOCK "DataLogCreate_DB"   // DB64
"DataLogCreate_SFB"
   // VAR_INPUT
   //    REQ : Bool;
   //    Records : UDInt;
   //    Format : UInt;
   //    Timestamp : UInt;
   //    "Name" : Variant;
   // END_VAR
   // VAR_OUTPUT
   //    DONE : Bool;
   //    BUSY : Bool;
   //    ERROR : Bool;
   //    STATUS : Word;
   // END_VAR
   // VAR_IN_OUT
   //    ID : DWord;
   //    Header : Variant;
   //    Data : Variant;
   // END_VAR
BEGIN
END_DATA_BLOCK

DATA_BLOCK "DataLogTimer01"   // DB63
{ S7_Optimized_Access := 'TRUE' }
"IEC_TIMER"
   // VAR
   //    PT : Time;
   //    ET : Time;
   //    IN : Bool;
   //    Q : Bool;
   // END_VAR
BEGIN
END_DATA_BLOCK

DATA_BLOCK "DataLogWrite_DB"   // DB65
"DataLogWrite_SFB"
   // VAR_INPUT
   //    REQ : Bool;
   // END_VAR
   // VAR_OUTPUT
   //    DONE : Bool;
   //    BUSY : Bool;
   //    ERROR : Bool;
   //    STATUS : Word;
   // END_VAR
   // VAR_IN_OUT
   //    ID : DWord;
   // END_VAR
BEGIN
END_DATA_BLOCK

DATA_BLOCK "DataLoggingDelay01"   // DB58
{ S7_Optimized_Access := 'TRUE' }
"IEC_TIMER"
   // VAR
   //    PT : Time;
   //    ET : Time;
   //    IN : Bool;
   //    Q : Bool;
   // END_VAR
BEGIN
END_DATA_BLOCK

DATA_BLOCK "Door_Closed_Delay"   // DB2
{ S7_Optimized_Access := 'TRUE' }
"IEC_TIMER"
   // VAR
   //    PT : Time;
   //    ET : Time;
   //    IN : Bool;
   //    Q : Bool;
   // END_VAR
BEGIN
END_DATA_BLOCK

DATA_BLOCK "DumbTimer"   // DB19
{ S7_Optimized_Access := 'TRUE' }
"IEC_TIMER"
   // VAR
   //    PT : Time;
   //    ET : Time;
   //    IN : Bool;
   //    Q : Bool;
   // END_VAR
BEGIN
END_DATA_BLOCK

DATA_BLOCK "Error_reset_again_timer"   // DB16
{ S7_Optimized_Access := 'TRUE' }
"IEC_TIMER"
   // VAR
   //    PT : Time;
   //    ET : Time;
   //    IN : Bool;
   //    Q : Bool;
   // END_VAR
BEGIN
END_DATA_BLOCK

DATA_BLOCK "Green_Blink"   // DB54
{ S7_Optimized_Access := 'TRUE' }
"IEC_TIMER"
   // VAR
   //    PT : Time;
   //    ET : Time;
   //    IN : Bool;
   //    Q : Bool;
   // END_VAR
BEGIN
END_DATA_BLOCK

DATA_BLOCK "Heater_Safety"   // DB14
{ S7_Optimized_Access := 'TRUE' }
"IEC_TIMER"
   // VAR
   //    PT : Time;
   //    ET : Time;
   //    IN : Bool;
   //    Q : Bool;
   // END_VAR
BEGIN
END_DATA_BLOCK

DATA_BLOCK "IEC_Timer_0_DB_ErrorAck01"   // DB4
{ S7_Optimized_Access := 'TRUE' }
"IEC_TIMER"
   // VAR
   //    PT : Time;
   //    ET : Time;
   //    IN : Bool;
   //    Q : Bool;
   // END_VAR
BEGIN
END_DATA_BLOCK

DATA_BLOCK "IEC_Timer_0_DB_ErrorAck02"   // DB7
{ S7_Optimized_Access := 'TRUE' }
"IEC_TIMER"
   // VAR
   //    PT : Time;
   //    ET : Time;
   //    IN : Bool;
   //    Q : Bool;
   // END_VAR
BEGIN
END_DATA_BLOCK

DATA_BLOCK "IEC_Timer_HeaterTimerV2"   // DB6
{ S7_Optimized_Access := 'TRUE' }
"IEC_TIMER"
   // VAR
   //    PT : Time;
   //    ET : Time;
   //    IN : Bool;
   //    Q : Bool;
   // END_VAR
BEGIN
END_DATA_BLOCK

DATA_BLOCK "IR_Heater_Reduce_Peak"   // DB60
{ S7_Optimized_Access := 'TRUE' }
"IEC_TIMER"
   // VAR
   //    PT : Time;
   //    ET : Time;
   //    IN : Bool;
   //    Q : Bool;
   // END_VAR
BEGIN
END_DATA_BLOCK

DATA_BLOCK "Initial_Test_Sequence_Delay"   // DB80
{ S7_Optimized_Access := 'TRUE' }
"IEC_TIMER"
   // VAR
   //    PT : Time;
   //    ET : Time;
   //    IN : Bool;
   //    Q : Bool;
   // END_VAR
BEGIN
END_DATA_BLOCK

DATA_BLOCK "Initial_Test_Sequence_Pulse"   // DB79
{ S7_Optimized_Access := 'TRUE' }
"IEC_TIMER"
   // VAR
   //    PT : Time;
   //    ET : Time;
   //    IN : Bool;
   //    Q : Bool;
   // END_VAR
BEGIN
END_DATA_BLOCK

DATA_BLOCK "Initial_Test_sequence_Delay02"   // DB81
{ S7_Optimized_Access := 'TRUE' }
"IEC_TIMER"
   // VAR
   //    PT : Time;
   //    ET : Time;
   //    IN : Bool;
   //    Q : Bool;
   // END_VAR
BEGIN
END_DATA_BLOCK

DATA_BLOCK "MC_MoveJog_DB"   // DB21
"MC_MoveJog"
   // VAR_INPUT
   //    Axis : TO_SpeedAxis;
   //    JogForward : Bool;
   //    JogBackward : Bool;
   //    Velocity : Real;
   //    PositionControlled : Bool;
   // END_VAR
   // VAR_OUTPUT
   //    InVelocity : Bool;
   //    Busy : Bool;
   //    CommandAborted : Bool;
   //    Error : Bool;
   //    ErrorID : Word;
   //    ErrorInfo : Word;
   // END_VAR
   // VAR
   //    FB_ID : DInt;
   // END_VAR
BEGIN
END_DATA_BLOCK

DATA_BLOCK "MC_MoveRelative_DB"   // DB42
"MC_MoveRelative"
   // VAR_INPUT
   //    Axis : TO_PositioningAxis;
   //    Execute : Bool;
   //    Distance : Real;
   //    Velocity : Real;
   // END_VAR
   // VAR_OUTPUT
   //    Done : Bool;
   //    Busy : Bool;
   //    CommandAborted : Bool;
   //    Error : Bool;
   //    ErrorID : Word;
   //    ErrorInfo : Word;
   // END_VAR
   // VAR
   //    FB_ID : DInt;
   // END_VAR
BEGIN
END_DATA_BLOCK

DATA_BLOCK "MC_Power_DB"   // DB13
"MC_Power"
   // VAR_INPUT
   //    Axis : TO_Axis;
   //    Enable : Bool;
   //    StartMode : Int;
   //    StopMode : Int;
   // END_VAR
   // VAR_OUTPUT
   //    Status : Bool;
   //    Busy : Bool;
   //    Error : Bool;
   //    ErrorID : Word;
   //    ErrorInfo : Word;
   // END_VAR
   // VAR
   //    FB_ID : DInt;
   // END_VAR
BEGIN
END_DATA_BLOCK

DATA_BLOCK "MachineConnected_Delay01"   // DB87
{ S7_Optimized_Access := 'TRUE' }
"IEC_TIMER"
   // VAR
   //    PT : Time;
   //    ET : Time;
   //    IN : Bool;
   //    Q : Bool;
   // END_VAR
BEGIN
END_DATA_BLOCK

DATA_BLOCK "MachineConnected_Delay02"   // DB88
{ S7_Optimized_Access := 'TRUE' }
"IEC_TIMER"
   // VAR
   //    PT : Time;
   //    ET : Time;
   //    IN : Bool;
   //    Q : Bool;
   // END_VAR
BEGIN
END_DATA_BLOCK

DATA_BLOCK "Red_Blink"   // DB53
{ S7_Optimized_Access := 'TRUE' }
"IEC_TIMER"
   // VAR
   //    PT : Time;
   //    ET : Time;
   //    IN : Bool;
   //    Q : Bool;
   // END_VAR
BEGIN
END_DATA_BLOCK

DATA_BLOCK "Reset_Green_Blink"   // DB56
{ S7_Optimized_Access := 'TRUE' }
"IEC_TIMER"
   // VAR
   //    PT : Time;
   //    ET : Time;
   //    IN : Bool;
   //    Q : Bool;
   // END_VAR
BEGIN
END_DATA_BLOCK

DATA_BLOCK "Reset_Red_Blink"   // DB55
{ S7_Optimized_Access := 'TRUE' }
"IEC_TIMER"
   // VAR
   //    PT : Time;
   //    ET : Time;
   //    IN : Bool;
   //    Q : Bool;
   // END_VAR
BEGIN
END_DATA_BLOCK

DATA_BLOCK "Reset_error_timer"   // DB11
{ S7_Optimized_Access := 'TRUE' }
"IEC_TIMER"
   // VAR
   //    PT : Time;
   //    ET : Time;
   //    IN : Bool;
   //    Q : Bool;
   // END_VAR
BEGIN
END_DATA_BLOCK

DATA_BLOCK "Staclight_MachineMoving_Timer_0_DB"   // DB85
{ S7_Optimized_Access := 'TRUE' }
"IEC_TIMER"
   // VAR
   //    PT : Time;
   //    ET : Time;
   //    IN : Bool;
   //    Q : Bool;
   // END_VAR
BEGIN
END_DATA_BLOCK

DATA_BLOCK "Timer_Red_Green_Blink"   // DB49
{ S7_Optimized_Access := 'TRUE' }
"IEC_TIMER"
   // VAR
   //    PT : Time;
   //    ET : Time;
   //    IN : Bool;
   //    Q : Bool;
   // END_VAR
BEGIN
END_DATA_BLOCK

DATA_BLOCK "Timer_Red_Green_Blink_Reset"   // DB50
{ S7_Optimized_Access := 'TRUE' }
"IEC_TIMER"
   // VAR
   //    PT : Time;
   //    ET : Time;
   //    IN : Bool;
   //    Q : Bool;
   // END_VAR
BEGIN
END_DATA_BLOCK

DATA_BLOCK "UVLamp_SafetyTimer_0_DB"   // DB84
{ S7_Optimized_Access := 'TRUE' }
"IEC_TIMER"
   // VAR
   //    PT : Time;
   //    ET : Time;
   //    IN : Bool;
   //    Q : Bool;
   // END_VAR
BEGIN
END_DATA_BLOCK

DATA_BLOCK "X_OnDelay"   // DB34
{ S7_Optimized_Access := 'TRUE' }
"IEC_TIMER"
   // VAR
   //    PT : Time;
   //    ET : Time;
   //    IN : Bool;
   //    Q : Bool;
   // END_VAR
BEGIN
END_DATA_BLOCK

DATA_BLOCK "X_Pulse"   // DB35
{ S7_Optimized_Access := 'TRUE' }
"IEC_TIMER"
   // VAR
   //    PT : Time;
   //    ET : Time;
   //    IN : Bool;
   //    Q : Bool;
   // END_VAR
BEGIN
END_DATA_BLOCK

DATA_BLOCK "Y_OnDelay"   // DB36
{ S7_Optimized_Access := 'TRUE' }
"IEC_TIMER"
   // VAR
   //    PT : Time;
   //    ET : Time;
   //    IN : Bool;
   //    Q : Bool;
   // END_VAR
BEGIN
END_DATA_BLOCK

DATA_BLOCK "Y_Pulse"   // DB38
{ S7_Optimized_Access := 'TRUE' }
"IEC_TIMER"
   // VAR
   //    PT : Time;
   //    ET : Time;
   //    IN : Bool;
   //    Q : Bool;
   // END_VAR
BEGIN
END_DATA_BLOCK

DATA_BLOCK "Z1_ondelay"   // DB24
{ S7_Optimized_Access := 'TRUE' }
"IEC_TIMER"
   // VAR
   //    PT : Time;
   //    ET : Time;
   //    IN : Bool;
   //    Q : Bool;
   // END_VAR
BEGIN
END_DATA_BLOCK

DATA_BLOCK "Z1_pulse"   // DB25
{ S7_Optimized_Access := 'TRUE' }
"IEC_TIMER"
   // VAR
   //    PT : Time;
   //    ET : Time;
   //    IN : Bool;
   //    Q : Bool;
   // END_VAR
BEGIN
END_DATA_BLOCK

DATA_BLOCK "Z2_ondelay"   // DB26
{ S7_Optimized_Access := 'TRUE' }
"IEC_TIMER"
   // VAR
   //    PT : Time;
   //    ET : Time;
   //    IN : Bool;
   //    Q : Bool;
   // END_VAR
BEGIN
END_DATA_BLOCK

DATA_BLOCK "Z2_pulse"   // DB27
{ S7_Optimized_Access := 'TRUE' }
"IEC_TIMER"
   // VAR
   //    PT : Time;
   //    ET : Time;
   //    IN : Bool;
   //    Q : Bool;
   // END_VAR
BEGIN
END_DATA_BLOCK

DATA_BLOCK "ZAxis_RelativeMotion_D01"   // DB99
{ S7_Optimized_Access := 'TRUE' }
"IEC_TIMER"
   // VAR
   //    PT : Time;
   //    ET : Time;
   //    IN : Bool;
   //    Q : Bool;
   // END_VAR
BEGIN
END_DATA_BLOCK

DATA_BLOCK "Zaxis_RelativeMotion_D03"   // DB100
{ S7_Optimized_Access := 'TRUE' }
"IEC_TIMER"
   // VAR
   //    PT : Time;
   //    ET : Time;
   //    IN : Bool;
   //    Q : Bool;
   // END_VAR
BEGIN
END_DATA_BLOCK

DATA_BLOCK "Zaxis_Test_D01"   // DB44
{ S7_Optimized_Access := 'TRUE' }
"IEC_TIMER"
   // VAR
   //    PT : Time;
   //    ET : Time;
   //    IN : Bool;
   //    Q : Bool;
   // END_VAR
BEGIN
END_DATA_BLOCK

DATA_BLOCK "Zaxis_Test_D02"   // DB95
{ S7_Optimized_Access := 'TRUE' }
"IEC_TIMER"
   // VAR
   //    PT : Time;
   //    ET : Time;
   //    IN : Bool;
   //    Q : Bool;
   // END_VAR
BEGIN
END_DATA_BLOCK

DATA_BLOCK "Zaxis_Test_D03"   // DB98
{ S7_Optimized_Access := 'TRUE' }
"IEC_TIMER"
   // VAR
   //    PT : Time;
   //    ET : Time;
   //    IN : Bool;
   //    Q : Bool;
   // END_VAR
BEGIN
END_DATA_BLOCK
